FUNCTION Convert_UINT_TO_TOD : BOOL
VAR_INPUT
	in : UINT;
	out : REFERENCE TO TOD;
END_VAR
VAR
	converted : TOD;
END_VAR

converted := UINT_TO_TOD(in);

IF (TOD_TO_UINT(converted) <> in) THEN
	RETURN;
END_IF

out := converted;
Convert_UINT_TO_TOD := TRUE;

END_FUNCTION

(* stored: Version 1.1.0.1, ProductVersion 3.1.4024.12
   POU Convert_UINT_TO_TOD: Id {345690fa-abe9-4420-a8ce-87f70ac5cede}, SpecialFunc None *)
